PROGRAM PRG_OTHER
// A Program for implementing devices with minimal interaction.
VAR
    {attribute 'pytmc' := 'pv: PC1K0:XTES:FSW'}
    {attribute 'TcLinkTo' := .bFlowOk := TIIB[IM1K0-EL1004]^Channel 1^Input'}
    fbPC1K0FlowSwitch : FB_XTES_Flowswitch;

    {attribute 'pytmc' := 'pv: PC1K4:XTES:FSW'}
    {attribute 'TcLinkTo' := .bFlowOk := TIIB[FEE-K-PCW-FSW-EL1004]^Channel 2^Input'}
    fbPC1K4FlowSwitch : FB_XTES_Flowswitch;
END_VAR

fbPC1K0FlowSwitch();
fbPC1K4FlowSwitch();

END_PROGRAM

(* stored: Version 1.1.0.1, ProductVersion 3.1.4022.18
   POU PRG_OTHER: Id {404f3e80-89c9-4363-9ece-c8d5a2e49981}, SpecialFunc None *)
